(*
SPDX-FileCopyrightText: Â© 2026 Oleksandr Tiutyk <trofimich@gmail.com>
SPDX-License-Identifier: MIT
License: https://opensource.org/license/mit
*)

(*!
<summary>Internal helper program providing access to the current library namespace.</summary>
*)

{attribute 'no_explicit_call' := 'do not call this POU directly'}
PROGRAM INTERNAL CurrentNamespace
VAR
	{attribute 'hide'} 
	_NamespaceExtractor : NamespaceExtractor;
END_VAR

(*!
<summary>Gets a reference to the current library namespace string.</summary>
*)
{attribute 'monitoring' := 'call'}
PROPERTY Name : REFERENCE TO STRING
GET
Name REF= _NamespaceExtractor.CurrentNamespace;
END_GET
END_PROPERTY

END_PROGRAM

(* stored: Version 1.1.0.1
   POU CurrentNamespace: Id {2fd6ba25-d26d-4239-a1f1-e927ba32b15c}, SpecialFunc None
   Property Name: Id {e056e449-2e5f-43ff-85cc-c31271f3cdcd}
   Get Get: Id {dfe8c12a-dc3c-4c40-a563-7e4381a8857f} *)
